FUNCTION Porc_inicial_Bomba : BOOL
VAR_INPUT
	Caudal_SP:REAL;
	Caudal_Nominal:REAL;
END_VAR
VAR_OUTPUT
	PorcInicial:REAL;
END_VAR
VAR
END_VAR

IF Caudal_Nominal=0 THEN
	Caudal_Nominal:=1;
END_IF
PorcInicial:=(Caudal_SP/Caudal_Nominal)*100.0*1.0;

END_FUNCTION

(* stored: Version 1.1.0.1, ProductVersion 3.1.4024.12
   POU Porc_inicial_Bomba: Id {3ec0d559-6418-4e37-8c57-5a4fd3b348ba}, SpecialFunc None *)
